{attribute 'qualified_only'}
{attribute 'strict'}
TYPE ePowerOverride : 
(
    Global_control := 0,
    Local_control := 1
);
END_TYPE

(* stored: Version 1.1.0.1, ProductVersion 3.1.4024.6
   DUT ePowerOverride: Id {2079d13c-119f-0423-12e4-1fd7a51f6243} *)
